# EPICS StreamDevice protocol: streamDevice/lillaser.proto
# DolphinDAQ Lil Laser protocol file
# Built by examining examples at: https://paulscherrerinstitute.github.io/StreamDevice/protocol.html#gen
# And also by examining input/output formats at https://paulscherrerinstitute.github.io/StreamDevice/formats.html

Terminator = CR LF;

##### Common #####

info {
	ExtraInput = Ignore;
	out "*IDN?";
	in "%39c";
}

debug {
   ExtraInput = Ignore;
   out "%s";
   in "%39c";
}

TrigCountQ {
    out ":TRIGger:COUNt?";
    in "%u";
}

TrigCount {
    out ":TRIGger:COUNt %u";
    @init { TrigCountQ; }
}

#### Lil Laser #####

OutEnabledQ {
    out ":OUTPut:ENABled?";
    in "%b";
}

OutEnabled {
    out ":OUTPut:ENABled %b";
    @init { OutEnabledQ; }
}

PowersQ {
    out ":LASer:POWers:YARRay?";
    separator=",";
    in "%u";
}

Powers {
    out ":LASer:POWers:YARRay %u";
    separator=",";
    @init { PowersQ; }
}

PowersDtQ {
    out ":LASer:POWers:DT?";
    in "%u";
}

PowersNtQ {
    out ":LASer:POWers:NT?";
    in "%u";
}
